(* CODESYS project set_pwm_frequency.20190318.1.project

Project tree, tasks and I/O mapping:
  MIC7001 : Changsha Xiangji-ARM Cortex A9(xilinx zynq7000)-linux, Changsha Xiangji Hiden Technology Co.Ltd, version 3.5.10.40
    application Application
      libraries: CAA Types Extern, 3.5.10.0 (CAA Technical Workgroup); VisuDialogs, * (System); CAA Real Time Clock Extern, 3.5.10.0 (CAA Technical Workgroup); CAA Callback Extern, 3.5.11.0 (CAA Technical Workgroup); CAA Can Low Level Extern, 3.5.11.0 (CAA Technical Workgroup); CAA Can Low Level Imp Extern, 3.5.11.0 (CAA Technical Workgroup); SysMem, 3.5.12.0 (System); CAA Net Base Services, 3.5.12.0 (CAA Technical Workgroup); Standard, 3.5.12.0 (System); CAA SerialCom, 3.5.12.0 (CAA Technical Workgroup); CAA File, 3.5.12.0 (CAA Technical Workgroup); CAA DTUtil Extern, 3.5.12.0 (CAA Technical Workgroup); SysFile, 3.5.9.0 (System); SysTypes2 Interfaces, * (System)
      task Task (cyclic, interval 10 ms, priority 10) calls prg_main
      task VISU_TASK (cyclic, interval 100 ms, priority 31) calls VisuElems.Visu_Prg
      visualisation main
      program prg_main [ST]
      global variables GVL
      trace Trace111 (task Task): trace_val
      function fn_set_pwm_frequency [ST]
    SoftMotion General Axis Pool
    IoDrvMIC7001 : IoDrvMIC7001, Cyber-MI, version 19.1.1
        input  Application.prg_main.pwm_feedback : DWORD  // Ai53_Pwm-i0
        output Application.prg_main.pwm : DWORD  // PWM28-Pwmi00@C33
        unmapped channels: Ai00@C16, Ai01@C28, Ai02@C17, Ai03@C29, Ai04@C30, Ai05@C19, Ai06@C31, Ai07@C20, Ai08@C18, Ai09@D18, Ai10@D20, Ai11@D31, Ai12@D19, Ai13@D30, Ai14@D29, Ai15@D17, Ai16@D28, Ai17@D16, Ai18-Do00@C25, Ai19-Do01@C24, Ai20-Do02@C13, Ai21-Do03@C01, Ai22-Do04@C03, Ai23-Do05@C04, Ai24-Do06@C05, Ai25-Do07@C06, Ai26-Do08@C08, Ai27-Do09@C09, Ai28-Do10@C10, Ai29-Do11@C11, Ai30-Do12@D34, Ai31-Do13@D35, Ai32-Do14@D23, Ai33-Do15@D12, Ai34-Do16@D10, Ai35-Do17@D09, Ai36-Do18@D08, Ai37-Do19@D07, Ai38-Do20@D05, Ai39-Do21@D04,
          Ai40-Do22@D03, Ai41-Do23@D02, Ai42-Do24@C23, Ai43-Do25@C35, Ai44-Do26@D24, Ai45-Do27@D13, Ai46-Ao00@C22, Ai47-Ao01@D14, Ai48_Pi02, Ai49_Out5V, Ai50_VCC, Ai51_VCC_L, Ai52_VCC_R, Ai54_Pwm-i1, Ai55_Pwm-i2, Ai56_Pwm-i3, Ai57_CPU-T, Ai58_G-x, Ai59_G-y, Ai60_G-z, Ai61-reserved, Ai62-IO-cntr, Ai63-CDS-cntr, Di00-Ai00@C16, Di01-Ai01@C28, Di02-Ai02@C17, Di03-Ai03@C29, Di04-Ai04@C30, Di05-Ai05@C19, Di06-Ai06@C31, Di07-Ai07@C20, Di08-Ai08@C18, Di09-Ai09@D18, Di10-Ai10@D20, Di11-Ai11@D31, Di12-Ai12@D19, Di13-Ai13@D30, Di14-Ai14@D29, Di15-Ai15@D17, Di16-Ai16@D28,
          Di17-Ai17@D16, Di18-Ai18@C25, Di19-Ai19@C24, Di20-Ai20@C13, Di21-Ai21@C01, Di22-Ai22@C03, Di23-Ai23@C04, Di24-Ai24@C05, Di25-Ai25@C06, Di26-Ai26@C08, Di27-Ai27@C09, Di28-Ai28@C10, Di29-Ai29@C11, Di30-Ai30@D34, Di31-Ai31@D35, Di32-Ai32@D23, Di33-Ai33@D12, Di34-Ai34@D10, Di35-Ai35@D09, Di36-Ai36@D08, Di37-Ai37@D07, Di38-Ai38@D05, Di39-Ai39@D04, Di40-Ai40@D03, Di41-Ai41@D02, Di42-Ai42@C23, Di43-Ai43@C35, Di44-Ai44@D24, Di45-Ai45@D13, Di46-Ai46@C22, Di47-Ai47@D14, Di48-Pi00@C15, Di49-Pi01@C14, Di50-Pi02@D22, Di51-Pi03@D21, Di52-reserved, Di53-reserved, Di54-reserved, Di55-reserved, Di56-reserved,
          Di57-reserved, Di58-reserved, Di59-reserved, Di60-reserved, Di61-reserved, Di62-reserved, Di63-reserved, Pi00-Di48@C15, Pi01-Di49@C14, Pi02-Di50@D22, Pi03-Di51@D21, Do00-Ai18@C25, Do01-Ai19@C24, Do02-Ai20@C13, Do03-Ai21@C01, Do04-Ai22@C03, Do05-Ai23@C04, Do06-Ai24@C05, Do07-Ai25@C06, Do08-Ai26@C08, Do09-Ai27@C09, Do10-Ai28@C10, Do11-Ai29@C11, Do12-Ai30@D34, Do13-Ai31@D35, Do14-Ai32@D23, Do15-Ai33@D12, Do16-Ai34@D10, Do17-Ai35@D09, Do18-Ai36@D08, Do19-Ai37@D07, Do20-Ai38@D05, Do21-Ai39@D04, Do22-Ai40@D03, Do23-Ai41@D02, Do24-Ai42@C23, Do25-Ai43@C35, Do26-Ai44@D24, Do27-Ai45@D13, Do28-Pwmi00@C33,
          Do29-Pwmi01@C34, Do30-Pwmi02@D25, Do31-Pwmi03@D26, PWM00@C25, PWM01@C24, PWM02@C13, PWM03@C01, PWM04@C03, PWM05@C04, PWM06@C05, PWM07@C06, PWM08@C08, PWM09@C09, PWM10@C10, PWM11@C11, PWM12@D34, PWM13@D35, PWM14@D23, PWM15@D12, PWM16@D10, PWM17@D09, PWM18@D08, PWM19@D07, PWM20@D05, PWM21@D04, PWM22@D03, PWM23@D02, PWM24@C23, PWM25@C35, PWM26@D24, PWM27@D13, PWM29-Pwmi01@C34, PWM30-Pwmi02@D25, PWM31-Pwmi03@D26, PWM_I_0@C33, PWM_I_1@C34, PWM_I_2@D25, PWM_I_3@D26, Ao00-Ai46@C22, Ao01-Ai47@D14,
          LED_run, LED_err, LED_usr, ctrl_ai_raw, ctrl_adjust, ctrl_adj0, ctrl_adj1, ctrl_adj2, ctrl_adj3, ctrl_adj4
  5ce3da45-db07-42e7-a21c-a00fff4ed8f6|C:\Users\Administrator\Desktop\robotview1.bmp
  5ce3da45-db07-42e7-a21c-a00fff4ed8f6|C:\Users\Administrator\Desktop\robotview2.bmp
  text list GlobalTextList
  5ce3da45-db07-42e7-a21c-a00fff4ed8f6|C:\Users\Administrator\Desktop\1129.bmp
  5ce3da45-db07-42e7-a21c-a00fff4ed8f6|C:\Users\Administrator\Desktop\robotview0.bmp
*)

// MIC7001/Application/GVL
VAR_GLOBAL
	trace_val:DWORD;
END_VAR

// MIC7001/Application/prg_main
PROGRAM prg_main  //主控制程序
VAR
	stat :DINT:=0;
	bRet :BOOL;
	pwm:DWORD;
	pwm_feedback:DWORD;
END_VAR


CASE stat OF
0:
	bRet := fn_set_pwm_frequency(port := 0, freq_hz := 100); //PORT C 所有PWM端口频率设置为100Hz
	IF bRet THEN
		stat := 5;
	END_IF
5:
	bRet := fn_set_pwm_frequency(port := 1, freq_hz := 300); //PORT D 所有PWM端口频率设置为300Hz
	IF bRet THEN
		stat := 10;
	END_IF
10:
END_CASE

gvl.trace_val := pwm_feedback;

END_PROGRAM

// MIC7001/Application/fn_set_pwm_frequency
FUNCTION fn_set_pwm_frequency : bool
VAR_INPUT
	port:DINT;
	freq_hz:DINT;
END_VAR
VAR
	filename_l :STRING := 'pwm_freq_l.txt';
	filename_r :STRING := 'pwm_freq_r.txt';
	filename:STRING(255);
	
	hFile: RTS_IEC_HANDLE := 0;
	udiPos:UDINT;
	udiOpenError: RTS_IEC_RESULT;
	udiWriteError: RTS_IEC_RESULT;
	udiByteWrite:LWORD;
	str:STRING(255);
END_VAR

fn_set_pwm_frequency := FALSE;
IF freq_hz < 50 THEN
	RETURN;
ELSIF freq_hz > 1000 THEN
	RETURN;
END_IF

IF port = 0 THEN 
	filename := filename_l;
ELSE
	filename := filename_r;
END_IF

hFile := sysfileopen(szFile := filename, am := sysfile.AM_WRITE, pResult := ADR(udiOpenError));
IF hFile = RTS_INVALID_HANDLE THEN
	RETURN;
END_IF

udiPos := SysFileSetPos(hFile:=hFile, ulOffset := 0);
str:= ANY_TO_STRING(freq_hz);
str := concat(str, ANY_TO_STRING('$N'));
udiByteWrite := sysfile.SysFileWrite(hFile := hFile,pbyBuffer := ADR(str),ulSize := ANY_TO_DWORD(len(str)), pResult := ADR(udiWriteError));
IF udiByteWrite < 1 THEN
	RETURN;
END_IF

fn_set_pwm_frequency := TRUE;

END_FUNCTION

// MIC7001/Application/main
VISUALIZATION main  // 2x2
END_VISUALIZATION
